// TwinCAT 3 PLC project Assignment_1_PS
// ProgramVersion: 3.1.4024.0
// libraries:
//   Tc2_Standard, * (Beckhoff Automation GmbH)
//   Tc2_System, * (Beckhoff Automation GmbH)
//   Tc3_Module, * (Beckhoff Automation GmbH)
//   VisuSymbols,3.5.10.0,System
// project tree:
//   / GlobalTextList.TcGTLO, PlcTask.TcTTO, Visualization Manager.TcVMO (not stored)
//   GVLs/ GVL.TcGVL
//   POUs/ Amazon.TcPOU, MAIN.TcPOU, PostNL.TcPOU, TrackAndTraceInfo.TcPOU
//   VISUs/ Visualization.TcVIS
// real-time tasks:
//   TASK PlcTask: cycle T#10ms, priority 20, ADS port 350

CONFIGURATION Assignment_1_PS
    RESOURCE PLC ON TwinCAT3
        TASK PlcTask(INTERVAL := T#10ms, PRIORITY := 20);
        PROGRAM MAIN WITH PlcTask : MAIN;
    END_RESOURCE
END_CONFIGURATION

// ---- GVLs/GVL.TcGVL
{attribute 'qualified_only'}
VAR_GLOBAL
	
	LED_BestellingGeplaatst  : BOOL;		//Led die aangeeft dat bestelling is geplaatst
	LED_BestellingGeleverd   : BOOL;		//Led die aangeeft dat bestelling is geleverd
	LED_PakketBijOHP		 : BOOL;		//Led die aangeeft dat pakket bij ophaalpunt ligt
	LED_BestellingIngepakt	 : BOOL;		//Led die aangeeft dat het pakket is ingepakt door de webshop
	LED_BestellingGesorteerd : BOOL;
	
	BT_BestellingPlaatsen	 : BOOL;		//Knop om bestelling te simuleren
	BT_Deurbel				 : BOOL;		//Knop die deurbel simuleert
	BT_DeurOpen				 : BOOL;		//Simuleert of deur open wordt gedaan
	BT_BestellingOpgehaald   : BOOL;		//Geeft aan wanneer klant bestelling ophaalt bij ophaalpunt
	BT_BestellingOphalen	 : BOOL;		//Knop die simuleert dat bestelling is opgehaald bij ophaalpunt
	BT_ToonStatus			 : BOOL;		//Laat status van bestelling zien zordra er op deze knop gedrukt wordt
	BT_BestellingIngepakt	 : BOOL;		//Knop die simuleert dat de beslling is ingepakt
	BT_Overhandigen			 : BOOL;		//Knop die simuleert dat pakket is overhandigd aan PostNL
	BT_PakketSorteren		 : BOOL;		//Knop die simuleert dat pakket is gesorteerd bij PostNL
 	
	TEMP_OhpOfBezorgen		 : BOOL;		//Tijdelijke variabele voor ophalen of bezorgen van pakket. Dit zodat het tijdens het proces niet aangepast kan worden
	TEMP_Overhandigen		 : BOOL; 		//TIjdelijke variabele voor overhandigen pakket naar PostNL. Dit zodat het tijdens het bezorg proces niet reset
	
	SW_OphalenOfBezorgen	 : BOOL;		//Geeft de klant de optie om pakket te laten bezorgen of op te halen bij ophaalpunt
	TX_PakketInfo			 : STRING;		//Geeft info over bestelling
	
	
	Reset					 : BOOL;		//Reset programma naar stap 0
END_VAR

// ---- POUs/MAIN.TcPOU
//Individuele eindopdracht Proces&Safety
//Jesse de Klein
//516392
//10-11-2024

PROGRAM MAIN
VAR
	
END_VAR

Amazon();
PostNL();

END_PROGRAM

// ---- POUs/Amazon.TcPOU
//Individuele eindopdracht Proces&Safety
//Jesse de Klein
//516392
//10-11-2024

PROGRAM Amazon
VAR
	stap 	  : INT;
	Timer_30s : TON;
END_VAR


CASE stap OF
	0:
	
END_CASE








(*CASE stap OF
	
	0:  //Stap 0: Bestelling nog niet geplaatst, alle waarde op 0
		Timer_30s(IN := FALSE);
		GVL.LED_BestellingGeplaatst := FALSE;
		GVL.LED_BestellingGeleverd  := FALSE;
		GVL.LED_PakketBijOHP		:= FALSE;
		
		//Schakelt naar stap 1 zodra bestelling wordt geplaatst
		IF GVL.BT_BestellingPlaatsen THEN
			stap := 1;
		END_IF
	
	
		
	1:	//Stap 1: Bestelling is geplaatst, wachten op deurbel 
		GVL.LED_BestellingGeplaatst := TRUE;
	
		//Geeft de klant de optie om pakket te laten bezorgen of zelf op te halen
		//Kiest de klant voor zelf ophalen zal het programma naar stap 4 gaan
		IF GVL.SW_OphalenOfBezorgen THEN
			stap := 4;
		END_IF
		
		IF GVL.BT_Deurbel THEN
			stap := 2;
		END_IF
		
		
		
	2:	//Stap 2: Bezorgen staat aan de deur en wacht tot deur open wordt gedaan 
		
		//Start timer. Wanneer de deur na 10 seconden nog niet open is zal het pakket naar het ophaalpunt worden gebracht
		Timer_30s(IN := TRUE, PT := T#10S);
		
		//Wacht tot deur open gaat
		IF GVL.BT_DeurOpen THEN
			Timer_30s(IN := FALSE);
			stap := 3;
			
		//Gaat de deur niet open wordt het pakken naar het ophaalpunt gebracht (stap 4)
		ELSIF Timer_30s.Q THEN
			TImer_30s(IN := FALSE);
			stap := 4;
		END_IF
		
		
	
	3:	//Stap 3: Pakket is bezorgd
		GVL.LED_BestellingGeleverd := TRUE;
		GVL.LED_PakketBijOHP := FALSE;
		
		
		
	4:	//Stap 4: Pakket ligt bij ophaalpunt
		GVL.LED_PakketBijOHP := TRUE;
		
		//Wanneer pakket wordt opgehaald gaat het programma naar stap 3
		IF GVL.BT_BestellingOphalen THEN
			stap := 3;
		END_IF			 
	
END_CASE


//Aanroepen functie voor het tonen van de status van het pakket
IF GVL.BT_ToonStatus THEN
	GVL.TX_PakketInfo := TrackAndTraceInfo(stap);
END_IF

//Reset het programma naar stap 0
IF GVL.Reset THEN
	stap := 0;
END_IF

*)

END_PROGRAM

// ---- POUs/PostNL.TcPOU
PROGRAM PostNL
VAR
END_VAR

END_PROGRAM

// ---- POUs/TrackAndTraceInfo.TcPOU
FUNCTION TrackAndTraceInfo : STRING
VAR_INPUT
	stap : INT;	//Input parameter, huidige stap
END_VAR

//Functie kijkt in welke stap het programma zich bevindt en op basis daarvan toont het de bijbehorende status
CASE stap OF
	0:	TrackAndTraceInfo := 'Wachten op bestelling.';
	1:	TrackAndTraceInfo := 'Bestelling geplaatst!';
	2:	TrackAndTraceInfo := 'Bezorger staat voor uw deur.';
	3:	TrackAndTraceInfo := 'Bestelling is in uw handen!';
	4:	TrackAndTraceInfo := 'Bestelling aanwezig bij ophaalpunt.';
	ELSE
		TrackAndTraceInfo := 'Status onbekend.';
END_CASE

END_FUNCTION

// ---- GlobalTextList.TcGTLO
TEXTLIST GlobalTextList
  913 = '%s'
  680 = 'Aanwezig'
  298 = 'Amazon'
  946 = 'Besstelling geplaatst'
  797 = 'Besstelling ingepakt'
  760 = 'Besstelling plaatsen'
  498 = 'Bestelling inpakken'
  106 = 'Bezorgd!'
  555 = 'Deur open'
  815 = 'Deurbel'
  225 = 'Gesorteerd'
  91 = 'Huis'
  112 = 'Laten bezorgen'
  481 = 'Ophaalpunt'
  757 = 'Ophalen'
  969 = 'Ophalen bij ophaalpunt'
  976 = 'Overhandigen -->'
  999 = 'PostNL'
  465 = 'Reset'
  526 = 'Sorteren'
  796 = 'Toon '
  28 = 'Toon pakket info'
  33 = 'Toon T&T info'
  171 = 'Toon T&T infoToon '
  930 = 'Toon T7T info'
  641 = 'Webwinkel'
END_TEXTLIST

// ---- VISUs/Visualization.TcVIS
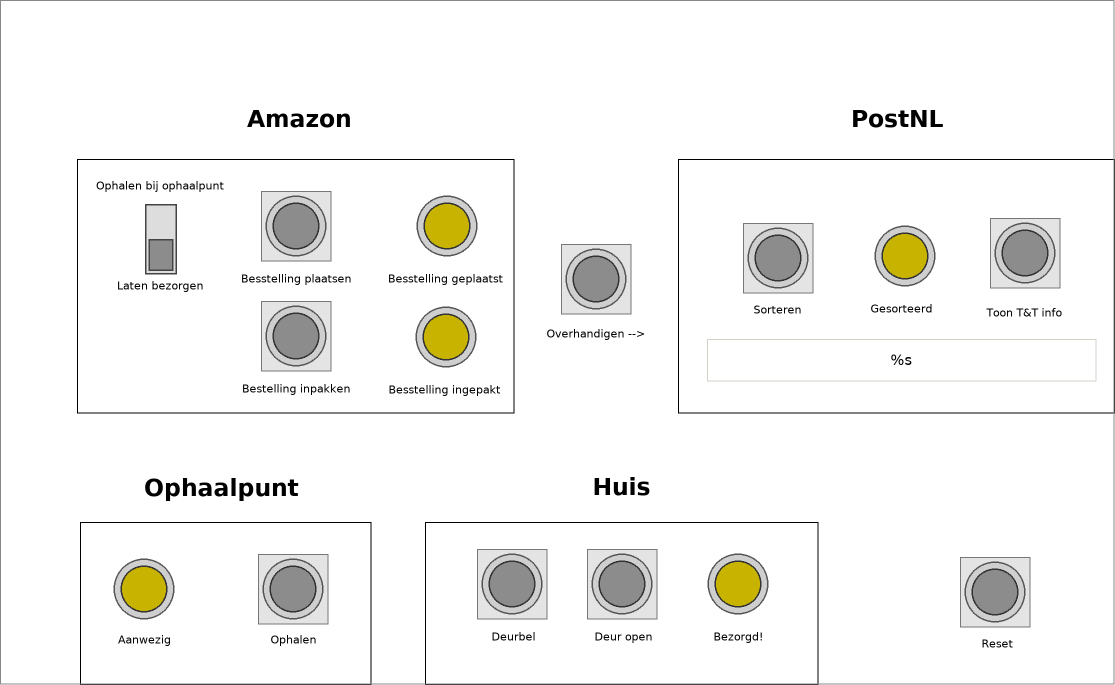
VISUALIZATION Visualization  // 1115x685
    RoundedRectangle (678,159 437x254)
    RoundedRectangle (80,522 291x163)
    RoundedRectangle (77,159 437x254)
    RoundedRectangle (425,522 393x163)
    Lamp1 (412,191 70x70), variable: GVL.LED_BestellingGeplaatst, style: Lamp-Lamp1-Yellow
    PushSwitch (477,549 70x70), variable: GVL.BT_Deurbel, behaviour: TAP, style: Switch-PushSwitch-Gray
    PushSwitch (960,557 70x70), variable: GVL.Reset, behaviour: TAP, style: Switch-PushSwitch-Gray
    PushSwitch (261,191 70x70), variable: GVL.BT_BestellingPlaatsen, behaviour: TAP, style: Switch-PushSwitch-Gray
    Label (237,264 119x30), "Besstelling plaatsen"
    Label (386,264 119x30), "Besstelling geplaatst"
    PushSwitch (587,549 70x70), variable: GVL.BT_DeurOpen, behaviour: TAP, style: Switch-PushSwitch-Gray
    Label (454,622 119x30), "Deurbel"
    Label (564,622 119x30), "Deur open"
    Label (938,629 119x30), "Reset"
    Label (217,104 165x30), "Amazon"
    Label (539,472 165x30), "Huis"
    Lamp1 (703,549 70x70), variable: GVL.LED_BestellingGeleverd, style: Lamp-Lamp1-Yellow
    Label (679,622 119x30), "Bezorgd!"
    Lamp1 (109,554 70x70), variable: GVL.LED_PakketBijOHP, style: Lamp-Lamp1-Yellow
    PushSwitch (258,554 70x70), variable: GVL.BT_BestellingOphalen, behaviour: TAP, style: Switch-PushSwitch-Gray
    Label (85,625 119x30), "Aanwezig"
    Label (234,625 119x30), "Ophalen"
    Label (139,473 165x30), "Ophaalpunt"
    DipSwitch (126,204 70x70), variable: GVL.SW_OphalenOfBezorgen, behaviour: TOGGLE, style: Switch-DipSwitch-Gray
    Label (101,271 119x30), "Laten bezorgen"
    Label (90,171 140x30), "Ophalen bij ophaalpunt"
    Label (467,473 245x30)
    PushSwitch (990,218 70x70), variable: GVL.BT_ToonStatus, behaviour: TAP, style: Switch-PushSwitch-Gray
    Textfield (707,339 389x42), "%s", text variable: GVL.TX_PakketInfo
    PushSwitch (561,244 70x70), variable: GVL.BT_Overhandigen, behaviour: TAP, style: Switch-PushSwitch-Gray
    Label (528,319 136x30), "Overhandigen -->"
    Label (815,104 165x30), "PostNL"
    PushSwitch (261,301 70x70), variable: GVL.BT_BestellingIngepakt, behaviour: TAP, style: Switch-PushSwitch-Gray
    Label (237,374 119x30), "Bestelling inpakken"
    Lamp1 (411,302 70x70), variable: GVL.LED_BestellingIngepakt, style: Lamp-Lamp1-Yellow
    Label (385,375 119x30), "Besstelling ingepakt"
    Label (965,298 119x30), "Toon T&T info"
    Lamp1 (870,221 70x70), variable: GVL.LED_BestellingGesorteerd, style: Lamp-Lamp1-Yellow
    Label (842,294 119x30), "Gesorteerd"
    PushSwitch (743,223 70x70), variable: GVL.BT_PakketSorteren, behaviour: TAP, style: Switch-PushSwitch-Gray
    Label (718,295 119x30), "Sorteren"
END_VISUALIZATION
